{attribute addProperty BoxType "AT2050-0501-0023"}
{attribute addProperty Id "A_0083_AT2050_5500_0016_AT2050_5500AT2050_C5E5984862678.25"}
{attribute addProperty CRC "1799803591"}
{attribute addProperty SizeInBites "626"}
{attribute addProperty SizeInBytes "78.25"}
TYPE A_0071_AT2050_0501_0023_AT2050_0501_6B46D2C7 EXTENDS AT2050_BA5A9548 :
STRUCT
	{attribute addProperty Name "A_0083_AT2050_5500_0016_AT2050_5500"}
	A_0083_AT2050_5500_0016_AT2050_5500 : AT2050_C5E59848;
END_STRUCT
END_TYPE

(* stored: Version 1.2.0.0, ProductVersion 3.1.4024.9
   DUT A_0071_AT2050_0501_0023_AT2050_0501_6B46D2C7: Id {38025bdb-6a75-4dbc-95a3-d512f095e90c} *)
